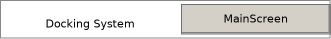
VISUALIZATION DockingStation  // 331x39
    Label (15,9 150x30), "Docking System"
    Button (181,4 150x30), "MainScreen"
        OnMouseClick: change screen: MainScreen
END_VISUALIZATION

(* stored: Version 1.1.0.1, ProductVersion 3.1.4024.12
   Visu DockingStation: Id {67f9a1b9-3dca-44e0-8245-e665cd9ce16d} *)
